TYPE HMIMessage :
STRUCT
	Channel	: DINT;
	Color	: DINT;
	Text	: T_MaxString;
	AltText	: T_MaxString;
END_STRUCT
END_TYPE

(* stored: Version 1.1.0.1, ProductVersion 3.1.4024.9
   DUT HMIMessage: Id {4d5d315b-a104-4365-9a4f-1c009095efa4} *)
